(* CoDeSys 2.3.9.62 project: GUI.pro *)
(* Libraries: Standard.lib, Iecsfc.lib 8.11.10 11:37:48, SYSLIBCALLBACK.LIB *)

(* PLC configuration (modules and I/O channels)
K-Bus [K_Bus] node 0, in %IB0 out %QB0
Internal Digital I/O [InternalDigIO] node 1, in %IB512 out %QB512
  Internal Digital Inputs [Internal_DIN] node 0, in %IB512 out %QB512
    DIN1 AT %IX2300.0 [BOOLOnX_I] Internal Digital Input Bit 1
    DIN2 AT %IX2300.1 [BOOLOnX_I] Internal Digital Input Bit 2
  Internal Digital Outputs [Internal_DOUT] node 1, in %IB513 out %QB512
    DOUT1 AT %QX2300.0 [BOOLOnX_Q] Internal Digital Output Bit 1
    DOUT2 AT %QX2300.1 [BOOLOnX_Q] Internal Digital Output Bit 2
Fieldbus variables [FB_VARS] node 3, in %IB0 out %QB0
Flag variables [FLAG_VARS] node 4, in %IB0 out %QB0
Modbus-Master [MB_MASTER] node 5, in %IB0 out %QB0
*)

(* Task configuration *)
TASK NewTask (PRIORITY := 15);
	mainTest();
END_TASK

(* Global variable list: Global_Variables *)
VAR_GLOBAL
	emergencyStopState : BOOL;
	motorIsOkay : BOOL;
	sikringIsOkay : BOOL;

	tapPC : BOOL
	pcTimer : INT;

	pedalsForward : BOOL;
	pedalsBack : BOOL;

	strenghtSlider : INT;
	rollSlider : INT;
	pitchSlider : INT;

	motorAngleDegrees0 : LREAL;
	motorAngleDegrees1: LREAL;
	motorAngleDegrees2: LREAL;

	innerOuterSlider : BOOL;
	innerOuterXOffset : INT;

	staticDynamicSlider : BOOL;
	staticDynamicXOffset : INT;
END_VAR

(* POU mainTest, ST *)
PROGRAM mainTest
VAR
	c : INT;
	tmp : LREAL;

	emergencyState : BOOL;

	angleFunction : ComputeMotorAngles;

	angle0 : LREAL;
	angle1: LREAL;
	angle2: LREAL;
	didBound: BOOL;
END_VAR
c := c + 1;
tmp := 5.0 / 2.0;

emergencyStopState := emergencyState;


innerOuterXOffset := 110 * BOOL_TO_INT(innerOuterSlider);
staticDynamicXOffset := 110 * BOOL_TO_INT(staticDynamicSlider);

angleFunction.roll := rollSlider / 2000.0;
angleFunction.pitch := pitchSlider / 2000.0;

angleFunction();

IF staticDynamicSlider THEN
	angle0 := angleFunction.angle0;
	angle1 := angleFunction.angle1;
	angle2 := angleFunction.angle2;
	didBound := angleFunction.didBound;
ELSE
	angle0 := 1.5708;
	angle1 := 1.5708;
	angle2 := 1.5708;
END_IF

motorAngleDegrees0 := 360.0 * angle0 / 6.28319;
motorAngleDegrees1 := 360.0 * angle1 / 6.28319;
motorAngleDegrees2 := 360.0 * angle2 / 6.28319;
END_PROGRAM

(* POU ComputeMotorAngles, ST *)
FUNCTION_BLOCK ComputeMotorAngles
VAR_INPUT
	roll : LREAL;
	pitch : LREAL;
END_VAR
VAR_OUTPUT
	angle0 : LREAL;
	angle1 : LREAL;
	angle2 : LREAL;

	didBound : BOOL;
END_VAR
VAR
	l : LREAL := 1.75;
	delta : LREAL;
	s0 : LREAL := 1.0;
	s1 : LREAL := 1.0;

	tmpVar : LREAL;

	p0 : LREAL;
	p1 : LREAL;
	p2 : LREAL;
END_VAR
delta := 0.03 * BOOL_TO_INT(innerOuterSlider) + 0.05;


tmpVar := l / 2 * ATAN(pitch / s1);
p1 :=delta + tmpVar;
p0 := delta - tmpVar;

p2 := delta - (l * SQRT(3) / 2) * ATAN(roll / s0);

p0 := -1.0 * (p0 - delta) / delta;
p1 := -1.0 * (p1 - delta) / delta;
p2 := -1.0 * (p2 - delta) / delta;

didBound := FALSE;

IF (p0 > 1.0) THEN
	p0 := 1.0;
	didBound := TRUE;
ELSIF (p0 < -1.0) THEN
	p0 := -1.0;
	didBound := TRUE;
END_IF


IF (p1 > 1.0) THEN
	p1 := 1.0;
	didBound := TRUE;
ELSIF (p1 < -1.0) THEN
	p1 := -1.0;
	didBound := TRUE;
END_IF

IF (p2 > 1.0) THEN
	p2 := 1.0;
	didBound := TRUE;
ELSIF (p2 < -1.0) THEN
	p2 := -1.0;
	didBound := TRUE;
END_IF

angle0 := ACOS(p0);
angle1 := ACOS(p1);
angle2 := ACOS(p2);
END_FUNCTION_BLOCK

(* Visualisation GUI
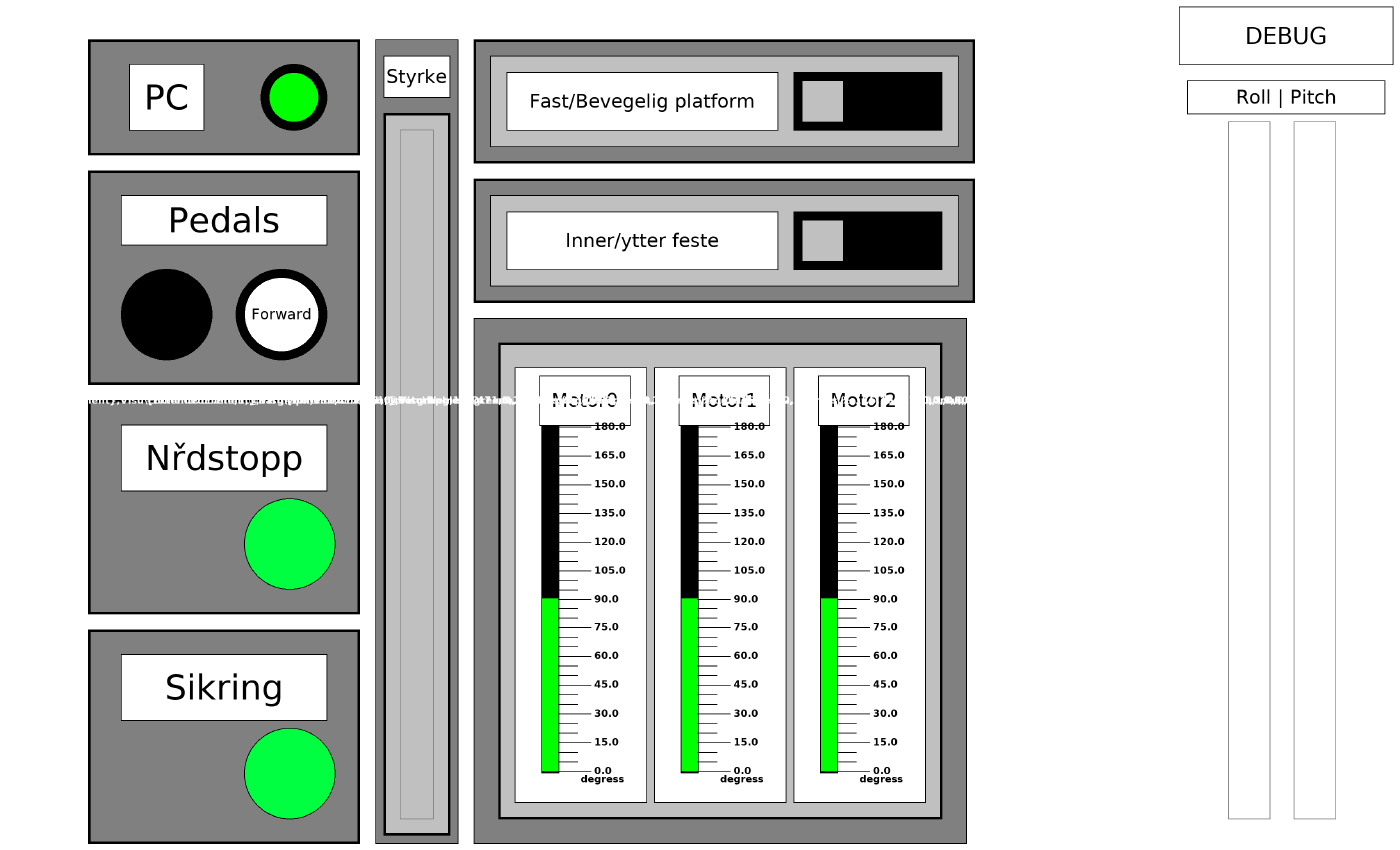
rounded rectangle at (90,520)-(341,601): text "Nřdstopp"
ellipse at (240,610)-(351,721): alarm colour if .emergencyStopState
rounded rectangle at (410,70)-(491,121): text "Styrke"
rounded rectangle at (90,800)-(341,881): text "Sikring"
ellipse at (240,890)-(351,1001): alarm colour if .sikringIsOkay
rectangle at (600,460)-(711,521): text "Motor0"
group at (570,490)-(751,961)
  rectangle at (0,0)-(1,1): text "{ExtendedElement},Visu\ElementDLL.ete,1,@Bargraph,181,471,0,1,0,motorAngleDegrees0,degress,%.1f,5,15,0,180,0,0,0,0,0,0,0,-13,16,700,Arial,0,255,0,255,0,0,0,0,1,0,0,0,0,,0,0,0,"
  rectangle at (31,228)-(49,426): alarm colour if (motorAngleDegrees0) < 0; top ((motorAngleDegrees0 * 1.0) - 90)  * -2.2
  rectangle at (88,415)-(168,436): text "0.0"
  rectangle at (88,382)-(168,403): text "15.0"
  rectangle at (88,349)-(168,370): text "30.0"
  rectangle at (88,316)-(168,337): text "45.0"
  rectangle at (88,283)-(168,304): text "60.0"
  rectangle at (88,250)-(168,271): text "75.0"
  rectangle at (88,218)-(168,239): text "90.0"
  rectangle at (88,185)-(168,206): text "105.0"
  rectangle at (88,152)-(168,173): text "120.0"
  rectangle at (88,119)-(168,140): text "135.0"
  rectangle at (88,86)-(168,107): text "150.0"
  rectangle at (88,53)-(168,74): text "165.0"
  rectangle at (88,20)-(168,41): text "180.0"
  rectangle at (50,427)-(148,443): text "degress"
rectangle at (770,460)-(881,521): text "Motor1"
group at (740,490)-(921,961)
  rectangle at (0,0)-(1,1): text "{ExtendedElement},Visu\ElementDLL.ete,1,@Bargraph,181,471,0,1,0,motorAngleDegrees1,degress,%.1f,5,15,0,180,0,0,0,0,0,0,0,-13,16,700,Arial,0,255,0,255,0,0,0,0,1,0,0,0,0,,0,0,0,"
  rectangle at (31,228)-(49,426): alarm colour if (motorAngleDegrees1) < 0; top ((motorAngleDegrees1 * 1.0) - 90)  * -2.2
  rectangle at (88,415)-(168,436): text "0.0"
  rectangle at (88,382)-(168,403): text "15.0"
  rectangle at (88,349)-(168,370): text "30.0"
  rectangle at (88,316)-(168,337): text "45.0"
  rectangle at (88,283)-(168,304): text "60.0"
  rectangle at (88,250)-(168,271): text "75.0"
  rectangle at (88,218)-(168,239): text "90.0"
  rectangle at (88,185)-(168,206): text "105.0"
  rectangle at (88,152)-(168,173): text "120.0"
  rectangle at (88,119)-(168,140): text "135.0"
  rectangle at (88,86)-(168,107): text "150.0"
  rectangle at (88,53)-(168,74): text "165.0"
  rectangle at (88,20)-(168,41): text "180.0"
  rectangle at (50,427)-(148,443): text "degress"
rectangle at (940,460)-(1051,521): text "Motor2"
group at (910,490)-(1091,961)
  rectangle at (0,0)-(1,1): text "{ExtendedElement},Visu\ElementDLL.ete,1,@Bargraph,181,471,0,1,0,motorAngleDegrees2,degress,%.1f,5,15,0,180,0,0,0,0,0,0,0,-13,16,700,Arial,0,255,0,255,0,0,0,0,1,0,0,0,0,,0,0,0,"
  rectangle at (31,228)-(49,426): alarm colour if (motorAngleDegrees2) < 0; top ((motorAngleDegrees2 * 1.0) - 90)  * -2.2
  rectangle at (88,415)-(168,436): text "0.0"
  rectangle at (88,382)-(168,403): text "15.0"
  rectangle at (88,349)-(168,370): text "30.0"
  rectangle at (88,316)-(168,337): text "45.0"
  rectangle at (88,283)-(168,304): text "60.0"
  rectangle at (88,250)-(168,271): text "75.0"
  rectangle at (88,218)-(168,239): text "90.0"
  rectangle at (88,185)-(168,206): text "105.0"
  rectangle at (88,152)-(168,173): text "120.0"
  rectangle at (88,119)-(168,140): text "135.0"
  rectangle at (88,86)-(168,107): text "150.0"
  rectangle at (88,53)-(168,74): text "165.0"
  rectangle at (88,20)-(168,41): text "180.0"
  rectangle at (50,427)-(148,443): text "degress"
rounded rectangle at (560,260)-(891,331): text "Inner/ytter feste"
rounded rectangle at (920,270)-(971,321): toggles .innerOuterSlider; x offset .innerOuterXOffset
rounded rectangle at (560,90)-(891,161): text "Fast/Bevegelig platform"
rounded rectangle at (920,100)-(971,151): toggles .staticDynamicSlider; x offset .staticDynamicXOffset
rectangle at (1380,10)-(1641,81): text "DEBUG"
rectangle at (1390,100)-(1631,141): text "Roll | Pitch"
rounded rectangle at (100,80)-(191,161): text "PC"
rounded rectangle at (90,240)-(341,301): text "Pedals"
ellipse at (240,340)-(331,431): text "Forward"; alarm colour if .emergencyStopState
ellipse at (270,90)-(331,151): taps .tapPC
137 more shapes without text or variables
7 elements of other kinds (tables, trends, ...) not read
*)
